{attribute 'linkalways'} 
{attribute 'no_explicit_call' := 'This FB is a CLASS and must be accessed using methods or properties'}
{attribute 'enable_dynamic_creation'}
FUNCTION_BLOCK _ETcVnKnn EXTENDS EnumDatatypeBase
VAR
	localData : ETcVnKnn;
	activeData : REFERENCE TO ETcVnKnn;
	enumBaseDatatype : _UDINT(localData);
END_VAR

METHOD PRIVATE AddLocalEnumeration
VAR_INPUT
	Enumeration : T_MAXSTRING;
	Value : ETcVnKnn;
END_VAR
AddEnumeration(Enumeration, Value);
END_METHOD

PROPERTY PUBLIC Address : PVOID
GET
Address := ADR(activeData);
END_GET
END_PROPERTY

METHOD PUBLIC ClearReference
VAR_INPUT
END_VAR
activeData REF= localData;
SetBaseDatatypeReference();
END_METHOD

METHOD PUBLIC Clone : I_Datatype
VAR
    pClone : POINTER TO _ETcVnKnn;
END_VAR
pClone := __NEW(_ETcVnKnn(InitialValue := Value));
Clone := pClone^;
END_METHOD

METHOD FB_init : BOOL
VAR_INPUT
	bInitRetains : BOOL; // if TRUE, the retain variables are initialized (warm start / cold start)
	bInCopyCode : BOOL;  // if TRUE, the instance afterwards gets moved into the copy code (online change)
	InitialValue : ETcVnKnn;
END_VAR
localData := InitialValue;
AddBaseDatatype(enumBaseDatatype);
ClearReference();

AddLocalEnumeration('TCVN_KNN_CLASSIFIER', ETcVnKnn.TCVN_KNN_CLASSIFIER);
AddLocalEnumeration('TCVN_KNN_NOVELTY_DETECTOR', ETcVnKnn.TCVN_KNN_NOVELTY_DETECTOR);
AddLocalEnumeration('TCVN_KNN_REGRESSOR', ETcVnKnn.TCVN_KNN_REGRESSOR);
END_METHOD

PROPERTY PUBLIC Identifier : T_MAXSTRING
GET
Identifier := 'ETcVnKnn';
END_GET
END_PROPERTY

METHOD IsEnumeratorValueEqual : BOOL
VAR_INPUT
	Enumerator : I_KeyValueForwardEnumerator;
END_VAR
VAR
	storedValue : ETcVnKnn;
END_VAR
IF NOT Enumerator.TryGet(storedValue) THEN
	RETURN;
END_IF

IsEnumeratorValueEqual := storedValue = activeData;
END_METHOD

METHOD PUBLIC MakeReferenceTo
VAR_INPUT
	ReferenceTarget : REFERENCE TO ETcVnKnn;
END_VAR
activeData REF= ReferenceTarget;
SetBaseDatatypeReference();
END_METHOD

METHOD PROTECTED SetBaseDatatypeReference
VAR_INPUT
END_VAR
enumBaseDatatype.MakeReferenceTo(activeData);
END_METHOD

PROPERTY PUBLIC Size : UDINT
GET
Size := SIZEOF(activeData);
END_GET
END_PROPERTY

METHOD TryMakeReferenceTo : BOOL
VAR_INPUT
	Target : I_Datatype;
END_VAR
VAR
	targetAsEnum : I_EnumDatatype;
	pTargetData : POINTER TO ETcVnKnn;
END_VAR
IF NOT Target.TryResolveAsEnumDatatype(targetAsEnum) THEN
	RETURN;
END_IF

IF targetAsEnum.Identifier <> Identifier THEN
	RETURN;
END_IF

pTargetData := Target.Address;
activeData REF= pTargetData^;
SetBaseDatatypeReference();
TryMakeReferenceTo := TRUE;
END_METHOD

PROPERTY PUBLIC Value : ETcVnKnn
GET
Value := activeData;
END_GET
SET
activeData := Value;
END_SET
END_PROPERTY

END_FUNCTION_BLOCK

(* stored: Version 1.1.0.1
   POU _ETcVnKnn: Id {f5c9655b-a1b9-4f88-b247-0b0bbbebe22a}, SpecialFunc None
   Folder Constructor: Id {aecf6b97-d50f-4985-a052-de1c44235cb9}
   Folder Private: Id {ae1c3205-a8df-4912-a600-cfa17aa2acf8}
   Folder Protected: Id {b6ebaff3-01da-4814-91cf-41c58a47c371}
   Method AddLocalEnumeration: Id {d2650ab9-6ecf-4a51-bdcf-730116f693ab}
   Property Address: Id {ee273b1a-7458-486b-a68d-ac3a6bcbdac4}
   Get Get: Id {09704946-2950-45ee-b506-f401b40aee5f}
   Method ClearReference: Id {88cdd417-e513-4612-800b-56303ab0673f}
   Method Clone: Id {4b3eda51-2075-4ffb-aaf4-5120a52e3a05}
   Method FB_init: Id {37e76beb-107d-4eae-8b09-5fa6f643e439}
   Property Identifier: Id {04224796-c920-4169-a4ee-97dd8957b612}
   Get Get: Id {b10a4721-706c-4fa7-9fef-a4fd157a9f26}
   Method IsEnumeratorValueEqual: Id {037e9303-7f73-49ca-8476-db4471a12c25}
   Method MakeReferenceTo: Id {d0dcaa6a-8b4c-4ce6-8675-8a6b47107064}
   Method SetBaseDatatypeReference: Id {23b1b64f-8856-4abd-9397-ceef6e7a8913}
   Property Size: Id {1308909f-8333-478c-b021-9d6b2ace2805}
   Get Get: Id {20954145-070b-4504-8ee2-67962686fb27}
   Method TryMakeReferenceTo: Id {5af6d00d-1d46-46f2-9b2b-8cd34155e3a4}
   Property Value: Id {33032d5e-cdcc-4715-b6c0-6b7074b7df7c}
   Get Get: Id {0f1092ef-6101-4c30-bf45-068783ebbbfd}
   Set Set: Id {dcaa36b1-61c2-4a93-a056-cd217ca179f6} *)
